# EPICS IOC start-up script: examples/test/PSI/ep1258.iocsh
#- mXsXXX naming
require ecmccfg v7_RC1, "NAMING=mXsXXX"

#- add slaves
${SCRIPTEXEC} ${ecmccfg_DIR}addSlave.cmd, "HW_DESC=EP1258, SLAVE_ID=5"
